(* CoDeSys 2.3 export: EvtCh16Tick32Bool8.EXP *)

(* POU core/evt/EvtCh16Tick32Bool8, ST *)
FUNCTION EvtCh16Tick32Bool8 : BOOL
VAR_INPUT
    Channel: UINT;
    Tick: UDINT;
    Value: BOOL;
END_VAR
VAR_IN_OUT
    Handle: LogBufferHandle;
END_VAR
VAR
    i: DINT;
    p1: POINTER TO BYTE;
    p2: POINTER TO BYTE;
    p3: POINTER TO UDINT;
END_VAR
i := GetNextWritePointer(11, Handle.BufferWritePointer, Handle.BufferReadPointer, Handle.BufferSize, Handle.BufferOverflow);
IF i >= 0 THEN

    p1 := Handle.BufferAddress + DINT_TO_DWORD(i);

    p1^ := START_FLAG;

    p1 := p1 + 1;
    p1^ := Handle.MagicByte;

    p1 := p1 + 1;
    p1^ := EVT_CH16_TICK32_BOOL8;

    p1 := p1 + 1;
    p2 := ADR(Channel);
    p1^ := p2^;

    p1 := p1 + 1;
    p2 := p2 + 1;
    p1^ := p2^;

    p3 := p1 + 1;
    p3^ := Tick;

    p1 := p1 + 5;
    p1^ := BOOL_TO_BYTE(Value);

    p1 := p1 + 1;
    p1^ := END_FLAG;

    Handle.BufferWritePointer := DWORD_TO_DINT(p1 - Handle.BufferAddress);

END_IF
END_FUNCTION
